// TIA Portal V17 export
// export: Created 2025-08-05T09:35:59.327424Z, ExportSetting WithDefaults, DisplayName Totally Integrated Automation Portal, DisplayVersion V17, DisplayName TIA Portal Openness, DisplayVersion V17, DisplayName TIA Portal Version Control Interface, DisplayVersion V17, DisplayName SINAMICS Startdrive Advanced, DisplayVersion V17, DisplayName SINAMICS Startdrive G130, G150, S120, S150, SINAMICS MV, S210, DisplayVersion V17, DisplayName SINAMICS Startdrive G110M, G120, G120C, G120D, G120P, G115D, DisplayVersion V17, DisplayName STEP 7 Professional, DisplayVersion V17, DisplayName STEP 7 Safety, DisplayVersion V17, DisplayName WinCC Advanced, DisplayVersion V17
VAR_GLOBAL   // PLC tag table "Standard IO"
   iScanner1 AT %I0.0 : "Scanner_Inputs";
   oScanner1 AT %Q0.0 : "Scanner_Outputs";
   iLaser1 AT %I48.0 : "YLS_Inputs";
   oLaser1 AT %Q32.0 : "YLS_Outputs";
END_VAR
